FUNCTION TryConvert_LREAL_TO_DINT : BOOL
VAR_INPUT
	in : LREAL;
	out : REFERENCE TO DINT;
END_VAR

IF in > DatatypeLimits.MAX_VALUE_OF_LREAL_WHICH_CAN_BE_HELD_IN_A_DINT THEN
	RETURN;
END_IF

IF in < DatatypeLimits.MIN_VALUE_OF_LREAL_WHICH_CAN_BE_HELD_IN_A_DINT THEN
	RETURN;
END_IF

out := LREAL_TO_DINT(in);
TryConvert_LREAL_TO_DINT := TRUE;

END_FUNCTION

(* stored: Version 1.1.0.1, ProductVersion 3.1.4024.12
   POU TryConvert_LREAL_TO_DINT: Id {b507ced7-2f28-4c61-aaaf-1b10efa90be1}, SpecialFunc None *)
